// TIA Portal V17 export
// export: Created 2025-03-07T09:16:36.9948107Z, ExportSetting WithDefaults, DisplayName Totally Integrated Automation Portal, DisplayVersion V17 Update 8, DisplayName TIA Portal Openness, DisplayVersion V17 Update 8, DisplayName TIA Portal Version Control Interface, DisplayVersion V17, DisplayName SINAMICS Startdrive Advanced, DisplayVersion V17 SP2, DisplayName SINAMICS Startdrive G110M, G120, G120C, G120D, G120P, G115D, DisplayVersion V17 SP2, DisplayName SINAMICS Startdrive G130, G150, S120, S150, SINAMICS MV, S210, DisplayVersion V17 SP2, DisplayName STEP 7 Professional, DisplayVersion V17 Update 8, DisplayName SINUMERIK ONE STEP 7 Toolbox, DisplayVersion V17 Update 12, DisplayName SINUMERIK 840D sl STEP 7 Toolbox, DisplayVersion V17 Update 12, DisplayName STEP 7 Safety, DisplayVersion V17 Update 6, DisplayName WinCC Advanced, DisplayVersion V17 Update 8
ORGANIZATION_BLOCK "OB40 Hardware interrupt"   // OB40, LAD, HardwareInterrupt
{ S7_Optimized_Access := 'TRUE' }
VERSION : 0.1
// stored: AutoNumber true, IsIECCheckEnabled false, SetENOAutomatically false
   VAR_INPUT
      LADDR : HW_IO;   // Hardware identifier
      USI : Word;   // User structure identifier
      IChannel : USInt;   // Interrupt channel number
      EventType : Byte;   // EventType
      PointAddr : DWord;
   END_VAR
   VAR_TEMP
      FLAG : Variant;
   END_VAR
BEGIN

REGION Network 2
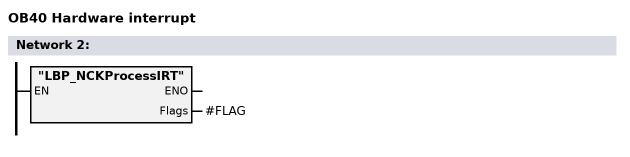
   RUNG wire#powerrail
      "LBP_NCKProcessIRT"(Flags => #FLAG)
   END_RUNG
   // the same network as SCL:
   "LBP_NCKProcessIRT"(Flags => #FLAG);
END_REGION
END_ORGANIZATION_BLOCK
